FUNCTION_BLOCK SynchPayload IMPLEMENTS I_Payload
VAR_INPUT
	bReleaseRequest : BOOL;
	bReleaseRequestReceived : BOOL;
	bRequestAck : BOOL;
	bRequestAckReceived : BOOL;
END_VAR
VAR_OUTPUT
END_VAR
VAR
END_VAR

END_FUNCTION_BLOCK

(* stored: Version 1.1.0.1, ProductVersion 3.1.4024.2
   POU SynchPayload: Id {0e6a2093-0152-4d23-96c0-2e9d1b1cc9da}, SpecialFunc None *)
